TYPE ZComUnit :
STRUCT
{region "Handling1"}
{IF NOT (defined (Handling1_disabled))}
  Handling1 : HandlingCom;
  {attribute 'ZId' := 'daa053b3-ae33-4567-9b11-72e6fc346262'}
{END_IF}
{endregion}
{region "Handling2"}
{IF NOT (defined (Handling2_disabled))}
  Handling2 : HandlingCom;
  {attribute 'ZId' := '686d4019-fd8f-49d1-bfb7-e2c5e589b8a3'}
{END_IF}
{endregion}
{attribute '__ZwPlcApplicationComUnitDeclaration__'} // Do not remove this attribute! It is used for code generation.
END_STRUCT
END_TYPE

(* stored: Version 1.1.0.1
   DUT ZComUnit: Id {e1525247-48b4-472d-9fd6-de4eb0da88da} *)
